VAR_GLOBAL
	
OP30_GIUDE_GRP_Manual_Axis: stManualModeAxis; 
OP30_GIUDE_GRP_ctrl: Servo_Control;	

SR30_Hori_servo_ctrl:Servo_Control;
SR30_Hori_servo_status:stManualModeAxis;

END_VAR

(* stored: Version 1.1.0.1, ProductVersion 3.1.4024.11
   GVL OP30_HMI_TAGS: Id {ec9ccb42-df5e-4fea-8cdf-5dae1a3820e1} *)
